{attribute 'OPC.UA.DA.StructuredType' := '1'}
TYPE ST_HVFAStorageState :
STRUCT
	fUpperTemperature 	: REAL;
	fLowerTemperature 	: REAL;
END_STRUCT
END_TYPE

(* stored: Version 1.1.0.1, ProductVersion 3.1.4024.10
   DUT ST_HVFAStorageState: Id {b98b734f-f795-4210-8193-4c96b5360b9a} *)
